ABB RobotStudio station: p2_sin.rspag

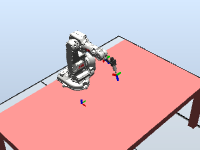
--- station ---
Station P2_paco (saved by RobotStudio 6.6.7701.1025)
Controller Sistema1
  mechanical unit ROB_1: IRB140_6_81_C_03, 6 joints, base frame (1250, 262.2, 836.07) mm, rotated rx 0 ry 0 rz 90 deg
Layout (positions relative to the parent item):
  - Mesa [part]
  - IRB140_6_81_C_03 [mechanism, from Robots\IRB140_6_81_C_G_03.rslib] at (1250, 262.2, 836.07) mm, rotated rx 0 ry 0 rz 90 deg; joint values [0, 0, 0, 0, 0.5236, 0] (rad or m)
  - MyTool [mechanism, from Libraries\myTool.rslib] at (1250, 768.49, 1515.57) mm, rotated rx -180 ry 60 rz -90 deg
Attachment: MyTool is attached to IRB140_6_81_C_03 / Link6

--- Backups/Sistema1/RAPID/TASK1/PROGMOD/CalibData.mod ---
MODULE CalibData
	PERS tooldata MyTool:=[TRUE,[[31.792631019,0,229.638935148],[0.945518576,0,0.325568154,0]],[1,[0,0,1],[1,0,0,0],0,0,0]];
	TASK PERS wobjdata placa:=[FALSE,TRUE,"",[[1500,600,850],[0.707106781,0,0,0.707106781]],[[0,0,0],[1,0,0,0]]];
ENDMODULE

--- Backups/Sistema1/RAPID/TASK1/PROGMOD/Module1.mod ---
MODULE Module1
    CONST robtarget Target_10:=[[351.468610021,249.99999759,-6.782975383],[0.01745192,-0.000000097,0.999847704,-0.000000068],[0,-3,1,0],[9E+09,9E+09,9E+09,9E+09,9E+09,9E+09]];
    CONST robtarget inicio:=[[351.468487273,250,523.21730631],[0.190808996,0,0.981627183,0],[0,0,0,0],[9E+09,9E+09,9E+09,9E+09,9E+09,9E+09]];
    CONST robtarget Target_20:=[[406.673861928,250.000001017,29.821690039],[0.017451896,-0.000000001,0.999847704,0.000000001],[0,-3,2,0],[9E+09,9E+09,9E+09,9E+09,9E+09,9E+09]];
    CONST robtarget abajo:=[[370.573303155,274.736754541,122.941555816],[0.034894192,-0.017441661,0.999238617,0.000609063],[0,0,-1,0],[9E+09,9E+09,9E+09,9E+09,9E+09,9E+09]];


    PROC sen()

    VAR num AMPY;
    VAR num AMPX;
    VAR num N;

    VAR robtarget p1;
    VAR robtarget p2;
    VAR robtarget p3;
    VAR robtarget p4;

    AMPY:=100;
    AMPX:=50;
    N:=1;

    p1:=Offs(Target_20,AMPX,AMPY,0);
    p2:=Offs(p1,-AMPX,AMPY,0);
    p3:=Offs(p2,-AMPX,AMPY,0);
    p4:=Offs(p3,AMPX,AMPY,0);

    FOR i FROM 1 TO N DO
        MoveJ inicio,v800,z200,MyTool\WObj:=placa;
        MoveL abajo,v1000,z100,MyTool\WObj:=placa;
        MoveC p1,p2,v100,fine,MyTool\WObj:=placa;
        MoveC p3,p4,v100,fine,MyTool\WObj:=placa;
        MoveC p3,p2,v100,fine,MyTool\WObj:=placa;
        MoveC p1,abajo,v100,z100,MyTool\WObj:=placa;

    ENDFOR
        MoveJ inicio,v1000,z200,MyTool\WObj:=placa;

    ENDPROC


    PROC main()
        sen;
    ENDPROC

ENDMODULE

--- Backups/Sistema1/RAPID/TASK1/PROGMOD/RsTempModule.mod ---
MODULE RsTempModule
PROC RsTempPath()
ENDPROC

ENDMODULE

--- Backups/Sistema1/RAPID/TASK1/SYSMOD/LINKEDM.sys ---
%%%
  VERSION:1
  LANGUAGE:ENGLISH
%%%

MODULE LINKEDM (SYSMODULE)

! FOLLOWER
!     Name of electronically linked follower axis used by operator at teach pendent.
      PERS string l_f_axis_name{5}       :=  ["",  "", "", "", ""];

!     Name of the mechanical unit for follower axis.
      PERS string l_f_mecunt_n{5}  :=  ["", "", "", "", ""];

!     Linked follower axis number in the mechanical unit (first axis in mech. unit is number 1).
      PERS num l_f_axis_no{5}      :=  [0,          0,   0,  0,  0];

! MASTER
!     Name of the mechanical unit for linked master axis.
      PERS string l_m_mecunt_n{5} :=  ["", "", "", "", ""];

!     Linked master axis number in the mechanical unit (first axis in mech. unit is number 1).
!     See axis number table in documentation for different master mechanical units.
      PERS num l_m_axis_no{5}     :=  [0,  0,  0,  0,  0];

! POSITION OFFSET
!     The increase of the allowed offset position between the master and follower
!     positions, used when starting AUTO mode. As soon as the offset is decreased
!     the old configurated parameter is used.
!     Example: 3 => the configurated value of allowed offset is increased 3 times.
      PERS num offset_ratio{5}       :=  [10,  10,   10,  10,  10];

! SPEED RATIO
!     Speed_ratio used in AUTO and JOG modes [ very_slow   slow    normal    fast]
!     Value 1 = max allowed manual speed.
      CONST num speed_ratio {20}      := [0.01, 0.01, 0.01, 0.01, 0.01,
                                          0.05, 0.05, 0.05, 0.05, 0.05,
                                          0.20, 0.20, 0.20, 0.20, 0.20,
                                          1.00, 1.00, 1.00, 1.00, 1.00];

! STEP SIZE
!     Displacement position used in JOG mode for each activation of positive or
!     negative movement.                  [very_short    short   normal   long]
!     Unit degees or meter.
      CONST num displacement {20}     := [0.001, 0.001, 0.001, 0.001, 0.001,
                                          0.005, 0.005, 0.005, 0.005, 0.005,
                                          0.020, 0.020, 0.020, 0.020, 0.020,
                                          0.100, 0.100, 0.100, 0.100, 0.100];


!-------------------------------------------------------------
 PROC Linked_m ()
      Linked_m_exe ;
 ENDPROC
ENDMODULE
